# EPICS autosave request: IOCs/MS_DAQ/MSApp/Db/MS_TwoThetaTemp_settings.req
# This file is used by autosave to determine what PVs to save (currently, autosave not used)
# It is also used by MS DAQ to determine what PVs to create

# This file contains all of the PVs used by the twoThetaTemp class.

####################
# Diffractometer Control
####################

$(P)$(R)TwoThetaMotorName
$(P)$(R)TwoThetaSpeedPVName
$(P)$(R)SpinnerMotorName

####################
# Gas Blower
####################

$(P)$(R)TempSetPointPVName
$(P)$(R)TempSP:RBVPVName
$(P)$(R)TempReadbackPVName
$(P)$(R)TempRatePVName
